(* CoDeSys 2.3 export: REGISTERADDRESS.EXP *)

(* Data type in INT *)
TYPE RegisterAddress : INT;
END_TYPE
